Omron Sysmac Studio project ClockFB (Sysmac Studio 1.56.0.64011, StandardProject)
(* 指定周期ごとにON、OFFを繰り返す信号を出力するFBです。 *)

# Controller new_Controller_0: NX102-1220 version 1.64
Task PrimaryTask (priority 4, period or condition 1000): Sample

PROGRAM Sample
VAR
    Clock_ins : yuyuTds\Clock;
    EnableClk : BOOL;
    Clk : BOOL;
END_VAR

(* Section Section0: ladder, written here as Structured Text *)

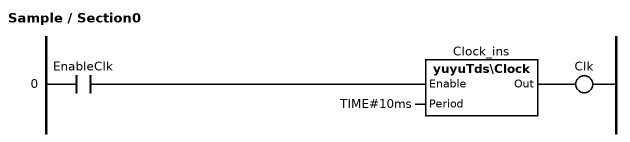
(* Rung 0 *)
Clock_ins(Enable := EnableClk, Period := TIME#10ms);
Clk := Clock_ins.Out;
END_PROGRAM

FUNCTION_BLOCK yuyuTds\Clock
(* 指定周期ごとにON、OFFを繰り返す信号を出力するFB *)
VAR
    EnableUp_ins : R_TRIG;  (* Enableの立上り *)
    wkCurrentCount : LINT;  (* 内部カウンタ *)
    wkTargetCount : LINT;  (* 内部カウンタ上限値 *)
END_VAR
VAR_INPUT
    Enable : BOOL;  (* 実行 *)
    Period : TIME;  (* クロック周期 *)
END_VAR
VAR_OUTPUT
    Out : BOOL;  (* 出力 *)
END_VAR
(*
【機能概要】
  指定した周期のクロック信号（ON、OFFを繰り返す信号）を出力するFB
    ・ Enableの立上りで、OutはTRUEになります。（出力ONから始まります）
    ・ 入力変数Periodは、タスク周期の倍数を指定してください。
	   倍数ではない場合、エラーになりませんが、出力の周期にズレが発生します。
  
【更新履歴】
  v1.0.0  24/04/06  初版
  
【GitHub】
  https://github.com/yuyuTds/ClockFB
*)

// □ Enableの立上りを監視
EnableUp_ins(Clk:=Enable);


// ■ 実行状態
IF Enable THEN
	
	// □ 初期処理（Enableの立上り）
	IF EnableUp_ins.Q THEN
		wkCurrentCount := 0;																													// 内部カウンタをリセット
		wkTargetCount := TimeToNanoSec(Period) / TimeToNanoSec(GetMyTaskInterval());					// 内部カウンタの上限値を設定（タスク周期数）
	END_IF;
	
	
	// □ 1：出力ON（周期前半）
	IF wkCurrentCount < (wkTargetCount / 2) THEN
		Out := TRUE;
	
	// □ 2：出力OFF（周期後半）
	ELSIF wkCurrentCount < wkTargetCount THEN
		Out := FALSE;
	END_IF;
	
	
	// □ カウントアップ
	wkCurrentCount := (wkCurrentCount + 1) MOD wkTargetCount;
	
	
// ■ 非実行状態
ELSE
	// □ 出力OFF
	Out := FALSE;
	
END_IF;
END_FUNCTION_BLOCK